PROGRAM MAIN
VAR
	Sensor1: BOOL;
	Sensor2: BOOL;
	Sensor3: BOOL;
	

	Motor1: BOOL;
	Motor2: BOOL;
	Motor3: BOOL;
	
	Sensor1On: BOOL;
	tonM2: TON;
	tonM1: TON;


END_VAR

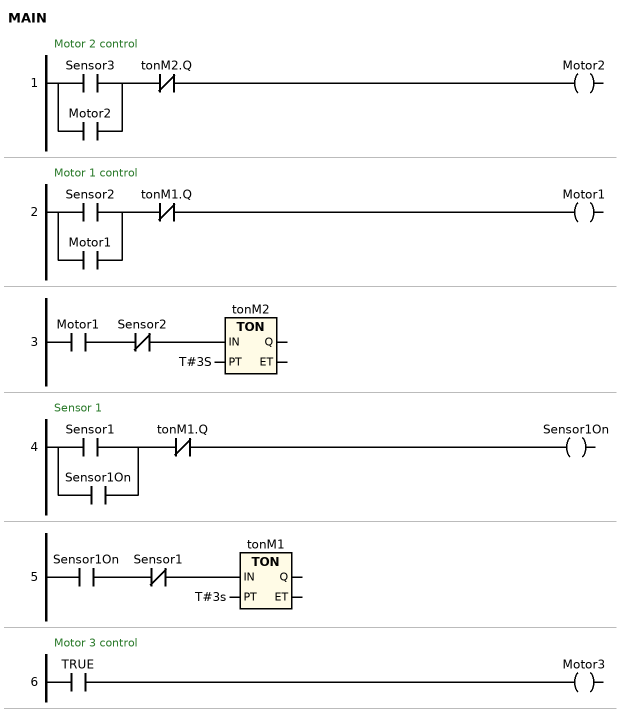
// NETWORK 1
// Motor 2 control
Motor2 := (Sensor3 OR Motor2) AND NOT tonM2.Q;

// NETWORK 2
// Motor 1 control
Motor1 := (Sensor2 OR Motor1) AND NOT tonM1.Q;

// NETWORK 3
tonM2(IN := Motor1 AND NOT Sensor2, PT := T#3S); // TON

// NETWORK 4
// Sensor 1
Sensor1On := (Sensor1 OR Sensor1On) AND NOT tonM1.Q;

// NETWORK 5
tonM1(IN := Sensor1On AND NOT Sensor1, PT := T#3s); // TON

// NETWORK 6
// Motor 3 control
Motor3 := TRUE;

END_PROGRAM

(* stored: Version 1.1.0.1, ProductVersion 3.1.4024.15
   POU MAIN: Id {9d5a4580-f23e-4666-bbce-b35e3e31b880}, SpecialFunc None *)
